TYPE SCodeCoverage_t :
STRUCT
	u16MaxPouIndex 	: UINT; (* speichert den größten Bausteinindex *)
	u16MaxLineIndex 	: UINT; (* Speichert den größten Zeilenindex*)
	aPou 					: ARRAY[1..PRG_TestCoverage.u32MaxPouIdx] OF ALines_t;
END_STRUCT
END_TYPE

(* stored: Version 1.1.0.1, ProductVersion 3.1.4024.9
   DUT SCodeCoverage_t: Id {c8bc135b-fcda-4943-82cb-c41edf0c3723} *)
